FUNCTION_BLOCK Tank_Fill EXTENDS _Tank_State
VAR
	_tonTimeout			: TON;
END_VAR

METHOD CanActivate : BOOL
CanActivate := _ctx.priv.smgr.Current = _ctx.state.iEnabled;
END_METHOD

METHOD OnExecute
_tonTimeout(IN := TRUE, PT := UDINT_TO_TIME(_ctx.hmi.nTimeout.val * 1000));
IF NOT _ctx.io.in.bEnable THEN
	_ctx.priv.smgr.Request(_ctx.state.iDisabled);
ELSIF _ctx.io.in.fLevel >= _ctx.hmi.fHighLevel.val THEN
	_ctx.priv.smgr.Request(_ctx.state.iEnabled);
ELSIF _tonTimeout.Q THEN
	_ctx.priv.smgr.Request(_ctx.state.iFault);
END_IF
END_METHOD

METHOD OnInit
_ctx.io.out.bInletValveOpen := TRUE;
_ctx.hmi.bResetButtonVis := FALSE;
_ctx.priv.IsFillable.Rise();
_tonTimeout(IN := FALSE);
END_METHOD

END_FUNCTION_BLOCK

(* stored: Version 1.1.0.1
   POU Tank_Fill: Id {956f5945-3487-4195-8577-fbca0c7baef1}, SpecialFunc None
   Method CanActivate: Id {a7eb6971-413b-4815-9fd0-5fa57c5fea70}
   Method OnExecute: Id {8e31315e-1c64-4547-9d14-8ff5304f8b20}
   Method OnInit: Id {400aacc0-abfd-4552-9899-8f5a53b857ba} *)
